FUNCTION_BLOCK CM_MOVITRAC_B EXTENDS CM_Base //IMPLEMENTS I_Motor_base
VAR_INPUT
	i_stSettings : ST_SettingsMOVITRAC_B_WithBrake;
	i_bIclkForward : BOOL := TRUE; //TRUE = interlocked
	i_bIclkBackward : BOOL := TRUE; //TRUE = interlocked
	
	i_ref_eCtrlState : REFERENCE TO E_CtrlState;
END_VAR
VAR
	// Inputs
	I_bStaReadyForOperation AT %I* : BOOL; // Drive is ready operation (no error)
	I_bStaMotorIsRunning AT %I* : BOOL; // Drive/motor is running
	
	// Outputs
	Q_bCmdReset AT %Q* : BOOL; // Command to reset drive.
	Q_bCmdEnable AT %Q* : BOOL; // Command to enable drive.
	Q_bCmdStartCW AT %Q* : BOOL; // Command start in clock-wise direction.
	Q_bCmdStartCCW AT %Q* : BOOL; // Command start in counter-clock-wise direction.
	
	Q_bCmdReleaseBrake AT %Q* : BOOL; // Command to release brake
	Q_nSetTargetSpeed AT %Q* : INT; // Target speed
	
	// Force outputs (IO-test functions)
	s_fbForceCmdReset : FB_ForceOutput;
	s_fbForceCmdEnable : FB_ForceOutput;
	s_fbForceCmdStartCW : FB_ForceOutput;
	s_fbForceCmdStartCCW : FB_ForceOutput;
	s_fbForceCmdReleaseBrake : FB_ForceOutput;
	s_fForceValueTargetSpeed : LREAL; //[0..100%]
	
	//Interlocks
	s_bIclkForward : BOOL;
	s_bIclkBackward : BOOL;
	
	// Requests
	s_bReqStop : BOOL;
	s_bReqStartForward : BOOL;
	s_bReqStartBackward : BOOL;
	s_bReqReleaseBrake : BOOL;
	s_bReqApplyBrake : BOOL;
	s_bReqReset : BOOL;
	
	// Commands
	s_bCmdEnable : BOOL;
	s_bCmdReset : BOOL;
	s_bCmdForward : BOOL;
	s_bCmdBackward : BOOL;
	s_bCmdReleaseBrake : BOOL;
		
	// States
	s_bStaReadyForOperation: BOOL;
	s_bStaDriveError: BOOL;
	s_bStaBrakeReleased : BOOL;
	s_bStaMotorStopped : BOOL;
	s_bStaWarning : BOOL;
	
	s_sInterlockedReasonForward : STRING; //External interlocked reason for clarifying reason
	s_sInterlockedReasonBackward : STRING; //External interlocked reason for clarifying reason
	
	// Setpoints
	s_fTargetSpeed : LREAL; // Target speed [mm/s]
	
	// Timers
	s_tofResetPulse : TOF;
	s_tonMotorStoppedDelay : TON;
	s_tonBrakeReleasedDelay : TON;
	
	// Alarms
	s_fbAlarmHandlerDriveError : FB_AlarmHandler;
	s_fbAlarmHandlerApplyingBrakeNotAllowed : FB_AlarmHandler;
	s_fbAlarmHandlerStartMotorNotAllowed : FB_AlarmHandler;
	s_fbAlarmHandlerMotorForwardInterlocked : FB_AlarmHandler;
	s_fbAlarmHandlerMotorBackwardInterlocked : FB_AlarmHandler;
	
	s_errDriveError : BOOL;
	s_wrnApplyingBrakeNotAllowed : BOOL;
	s_wrnStartMotorNotAllowed : BOOL;
	s_wrnMotorForwardInterlocked : BOOL;
	s_wrnMotorBackwardInterlocked : BOOL;
	
	//Hmi
	s_fbHmiBtnManualReleaseBrake: FB_HmiBtn;
	s_fbHmiBtnManualApplyBrake	: FB_HmiBtn;
	s_fbHmiBtnManualForward		: FB_HmiBtn;
	s_fbHmiBtnManualBackward	: FB_HmiBtn;
	s_fbHmiBtnManualStop		: FB_HmiBtn;
	s_fbHmiBtnManualReset		: FB_HmiBtn;
	
	s_fbHmiLedBrakeReleased		: FB_HmiLed;
	s_fbHmiLedMotorStopped		: FB_HmiLed;
	s_fbHmiLedDriveError		: FB_HmiLed;
	
	//Sequence
	eSeqMOVITRAC_B_WithBrake : E_SeqMOVITRAC_B_WithBrake;
	seqTimer : TON;
	seqPreStep : E_SeqMOVITRAC_B_WithBrake;
	s_sActStep : STRING;
	
END_VAR

VAR CONSTANT
	cMAX_INT_VALUE : INT := 32767;
END_VAR


SUPER^();

METHOD PROTECTED _m_Alarms : BOOL

IF NOT SUPER^._m_Alarms() THEN
	RETURN;
END_IF

// Set error bits
s_errDriveError := i_bReqEnable AND s_bStaDriveError;// AND NOT(i_bCmdReset);

// Interlock warnings
IF s_bIclkForward AND NOT(s_bStaMotorStopped) THEN	
	s_wrnMotorForwardInterlocked := TRUE;
	m_Stop();
ELSIF NOT(s_bIclkForward) OR i_bCmdReset THEN
	s_wrnMotorForwardInterlocked := FALSE;
END_IF

IF s_bIclkBackward AND NOT(s_bStaMotorStopped) THEN
	s_wrnMotorBackwardInterlocked := TRUE;
	m_Stop();
ELSIF NOT(s_bIclkBackward) OR i_bCmdReset THEN
	s_wrnMotorBackwardInterlocked := FALSE;
END_IF

// Alarm Handlers
s_fbAlarmHandlerDriveError(
	i_bStaActive := s_errDriveError,
	i_eAlarmLevel := E_AlarmLevel.Alarm,
	i_sAlarmText := CONCAT(i_sCmName, ': Drive - has error (check drive).'));
	
s_fbAlarmHandlerApplyingBrakeNotAllowed(
	i_bStaActive := s_wrnApplyingBrakeNotAllowed,
	i_eAlarmLevel := E_AlarmLevel.Warning,
	i_sAlarmText := CONCAT(i_sCmName, ': Brake - not allowed to be applied (motor not stopped).'));
	
s_wrnApplyingBrakeNotAllowed R= s_bStaMotorStopped;
	
s_fbAlarmHandlerStartMotorNotAllowed(
	i_bStaActive := s_wrnStartMotorNotAllowed,
	i_eAlarmLevel := E_AlarmLevel.Warning,
	i_sAlarmText := CONCAT(i_sCmName, ': Motor - not allowed to start (brake not released).'));
	
s_wrnStartMotorNotAllowed R= s_bStaBrakeReleased;
	
s_fbAlarmHandlerMotorForwardInterlocked(
	i_bStaActive := s_wrnMotorForwardInterlocked,
	i_eAlarmLevel := E_AlarmLevel.Warning,
	i_sAlarmText := CONCAT(i_sCmName, CONCAT(': Motor - interlocked to move forward, Reason: ',CONCAT(s_sInterlockedReasonForward, '.'))));
	//--i_sAlarmText := CONCAT(i_sCmName, CONCAT(': Motor - interlocked to move forward, Reason: ',CONCAT(i_fbInterlockConvFwd.p_sReason, '.'))));
	
s_fbAlarmHandlerMotorBackwardInterlocked(
	i_bStaActive := s_wrnMotorBackwardInterlocked,
	i_eAlarmLevel := E_AlarmLevel.Warning,
	i_sAlarmText := CONCAT(i_sCmName, CONCAT(': Motor - interlocked to move backward, Reason: ',CONCAT(s_sInterlockedReasonBackward, '.'))));
	//--i_sAlarmText := CONCAT(i_sCmName, CONCAT(': Motor - interlocked to move backward, Reason: ',CONCAT(i_fbInterlockConvBwd.p_sReason, '.'))));
	
// Alarm collector	
s_bStaError := 
	s_fbAlarmHandlerDriveError.q_bStaActive;

// Warning collector
s_bStaWarning := 
	s_fbAlarmHandlerApplyingBrakeNotAllowed.q_bStaActive
	OR s_fbAlarmHandlerStartMotorNotAllowed.q_bStaActive
	OR s_fbAlarmHandlerMotorForwardInterlocked.q_bStaActive
	OR s_fbAlarmHandlerMotorBackwardInterlocked.q_bStaActive;	
	
_m_Alarms := TRUE;
END_METHOD

METHOD PROTECTED _m_Devices : BOOL

IF NOT SUPER^._m_Devices() THEN
	RETURN;
END_IF

//Exception error
IF (s_bStaError OR NOT(i_bReqEnable))
	AND (eSeqMOVITRAC_B_WithBrake < E_SeqMOVITRAC_B_WithBrake.STOPPING) THEN
		eSeqMOVITRAC_B_WithBrake := E_SeqMOVITRAC_B_WithBrake.STOPPING;
END_IF 

seqTimer(
	IN := (eSeqMOVITRAC_B_WithBrake = seqPreStep),
	PT := T#3600S);
	
seqPreStep := eSeqMOVITRAC_B_WithBrake;

s_sActStep := TO_STRING(eSeqMOVITRAC_B_WithBrake);
	
CASE eSeqMOVITRAC_B_WithBrake OF
	
	E_SeqMOVITRAC_B_WithBrake.INIT:
		_m_ResetAllRequests();
	
		//Reset commands
		s_bCmdForward := FALSE;
		s_bCmdBackward := FALSE;	
		s_bCmdReleaseBrake := FALSE;
		s_bCmdReset := FALSE;
		s_bCmdEnable := FALSE;
		s_fTargetSpeed := 0;
		
		//Reset states
		s_bStaBrakeReleased := FALSE;
		s_bStaDriveError := FALSE;
		//s_bStaMotorStopped := FALSE;			written by inputs()
		//s_bStaReadyForOperation := FALSE;		written by inputs()
	
		eSeqMOVITRAC_B_WithBrake := E_SeqMOVITRAC_B_WithBrake.STOPPED; 
		
	E_SeqMOVITRAC_B_WithBrake.STOPPED:
		s_bStaBrakeReleased := FALSE;
		//--s_bStaMotorStopped := TRUE;			written by inputs()
		s_bReqStop := FALSE;
		s_bStaReadyForOperation := TRUE;
		
		IF (s_bReqReleaseBrake OR s_bReqStartForward OR s_bReqStartBackward) THEN
			eSeqMOVITRAC_B_WithBrake := E_SeqMOVITRAC_B_WithBrake.RELEASE_BRAKE;
		END_IF

		IF s_bReqApplyBrake THEN
			eSeqMOVITRAC_B_WithBrake := E_SeqMOVITRAC_B_WithBrake.APPLY_BRAKE;
		END_IF
		
		IF seqTimer.PT >= T#10S THEN
			s_bCmdEnable := FALSE;
		END_IF
			
	E_SeqMOVITRAC_B_WithBrake.RELEASE_BRAKE:
		s_bCmdReleaseBrake := TRUE;
		s_bReqReleaseBrake := FALSE;
		
		IF seqTimer.ET > i_stSettings.tBrakeReleasedDelay THEN
			s_bStaBrakeReleased := TRUE;
		END_IF
		
		IF s_bReqStop THEN
			eSeqMOVITRAC_B_WithBrake := E_SeqMOVITRAC_B_WithBrake.STOPPING;
		ELSIF s_bStaBrakeReleased AND s_bReqStartForward THEN
			s_bCmdEnable := TRUE;
			eSeqMOVITRAC_B_WithBrake := E_SeqMOVITRAC_B_WithBrake.MOVING_FORWARD;
		ELSIF s_bStaBrakeReleased AND s_bReqStartBackward THEN
			s_bCmdEnable := TRUE;
			eSeqMOVITRAC_B_WithBrake := E_SeqMOVITRAC_B_WithBrake.MOVING_BACKWARD;
		ELSIF s_bReqApplyBrake THEN
			eSeqMOVITRAC_B_WithBrake := E_SeqMOVITRAC_B_WithBrake.APPLY_BRAKE;
		END_IF
	
	E_SeqMOVITRAC_B_WithBrake.MOVING_FORWARD:
		s_bCmdForward := TRUE;
		s_bReqStartForward := FALSE;
		
		//--s_bStaMotorStopped := FALSE;		written by inputs()
		//s_fTargetSpeed is written by method 
	
		IF s_bReqStop THEN
			eSeqMOVITRAC_B_WithBrake := E_SeqMOVITRAC_B_WithBrake.STOPPING;
		END_IF
		
	E_SeqMOVITRAC_B_WithBrake.MOVING_BACKWARD:
		s_bCmdBackward := TRUE;
		s_bReqStartBackward := FALSE;
		
		//--s_bStaMotorStopped := FALSE;		//written by inputs()
		//s_fTargetSpeed is written by method 
	
		IF s_bReqStop THEN
			eSeqMOVITRAC_B_WithBrake := E_SeqMOVITRAC_B_WithBrake.STOPPING;
		END_IF
	
	E_SeqMOVITRAC_B_WithBrake.STOPPING:
		s_bCmdForward := FALSE;
		s_bCmdBackward := FALSE;
		s_bReqStop := FALSE;
		
		IF s_bStaMotorStopped THEN
			eSeqMOVITRAC_B_WithBrake := E_SeqMOVITRAC_B_WithBrake.APPLY_BRAKE;
		END_IF
		
		//--IF seqTimer.ET > i_stSettings.tMotorStoppedDelay THEN
			//--s_bStaMotorStopped := TRUE;		//Written by inputs()
			//--eSeqMOVITRAC_B_WithBrake := E_SeqMOVITRAC_B_WithBrake.APPLY_BRAKE;
		//--END_IF	
	
	E_SeqMOVITRAC_B_WithBrake.APPLY_BRAKE:
		s_bCmdReleaseBrake := FALSE;
		s_bReqApplyBrake := FALSE;
		
		IF seqTimer.ET > i_stSettings.tBrakeReleasedDelay THEN
			s_bStaBrakeReleased := FALSE;
			
			IF (s_bStaError OR NOT(i_bReqEnable)) THEN
				eSeqMOVITRAC_B_WithBrake := E_SeqMOVITRAC_B_WithBrake.ERROR;
			ELSE
				_m_ResetAllRequests();
				eSeqMOVITRAC_B_WithBrake := E_SeqMOVITRAC_B_WithBrake.STOPPED;
			END_IF	
		END_IF
		
	E_SeqMOVITRAC_B_WithBrake.ERROR:
		s_bCmdReset := i_bCmdReset OR s_bReqReset;
		s_bReqReset := FALSE;
		
		IF (NOT(s_bStaError) AND i_bReqEnable) THEN
			eSeqMOVITRAC_B_WithBrake := E_SeqMOVITRAC_B_WithBrake.INIT;
		END_IF
		
END_CASE

_m_Devices := TRUE;
END_METHOD

METHOD PROTECTED _m_Hmi : BOOL

IF NOT SUPER^._m_Hmi() THEN
	RETURN;
END_IF

//Buttons
s_fbHmiBtnManualReleaseBrake();
s_fbHmiBtnManualApplyBrake();
s_fbHmiBtnManualForward();
s_fbHmiBtnManualBackward();
s_fbHmiBtnManualStop();
s_fbHmiBtnManualReset();

//Led
s_fbHmiLedBrakeReleased(i_bStaLed := s_bStaBrakeReleased);
s_fbHmiLedMotorStopped(i_bStaLed := s_bStaMotorStopped);
s_fbHmiLedDriveError(i_bStaLed := s_bStaDriveError);
(*
{warning '#TODO: Add manual control from hmi'}
CASE i_eCtrlMode OF

	E_CtrlMode.IDLE..
	E_CtrlMode.AUTOMATIC:
		s_fbHmiBtnManualReleaseBrake.p_bStaVisible := FALSE;
		s_fbHmiBtnManualReleaseBrake.p_bStaEnabled := FALSE;
		
		s_fbHmiBtnManualApplyBrake.p_bStaVisible := FALSE;
		s_fbHmiBtnManualApplyBrake.p_bStaEnabled := FALSE;
		
		s_fbHmiBtnManualForward.p_bStaVisible := FALSE;
		s_fbHmiBtnManualForward.p_bStaEnabled := FALSE;
		
		s_fbHmiBtnManualBackward.p_bStaVisible := FALSE;
		s_fbHmiBtnManualBackward.p_bStaEnabled := FALSE;
		
		s_fbHmiBtnManualStop.p_bStaVisible := FALSE;
		s_fbHmiBtnManualStop.p_bStaEnabled := FALSE;
		
		s_fbHmiBtnManualReset.p_bStaVisible := FALSE;
		s_fbHmiBtnManualReset.p_bStaEnabled := FALSE;
	
	E_CtrlMode.MANUAL:
		//Is het de bedoeling om op deze plekken de hmi knoppen aan te sturen, OF moet dat gedaan worden in METHOD hmi?
		s_fbHmiBtnManualReleaseBrake.p_bStaVisible := TRUE;
		s_fbHmiBtnManualReleaseBrake.p_bStaEnabled := i_bReqEnable;
		
		s_fbHmiBtnManualApplyBrake.p_bStaVisible := TRUE;
		s_fbHmiBtnManualApplyBrake.p_bStaEnabled := i_bReqEnable AND s_bStaMotorStopped;
		
		s_fbHmiBtnManualForward.p_bStaVisible := TRUE;
		s_fbHmiBtnManualForward.p_bStaEnabled := i_bReqEnable AND s_bStaMotorStopped (*AND s_bStaBrakeReleased*) AND NOT(i_bIclkForward);
		
		s_fbHmiBtnManualBackward.p_bStaVisible := TRUE;
		s_fbHmiBtnManualBackward.p_bStaEnabled := i_bReqEnable AND s_bStaMotorStopped (*AND s_bStaBrakeReleased*) AND NOT(i_bIclkBackward);
		
		s_fbHmiBtnManualStop.p_bStaVisible := TRUE;
		s_fbHmiBtnManualStop.p_bStaEnabled := TRUE;
		
		s_fbHmiBtnManualReset.p_bStaVisible := TRUE;
		s_fbHmiBtnManualReset.p_bStaEnabled := TRUE;
		
		IF s_fbHmiBtnManualReleaseBrake.p_osrBtnPress THEN
			m_ReleaseBrake();
		END_IF
	
		IF s_fbHmiBtnManualApplyBrake.p_osrBtnPress THEN
			m_ApplyBrake();
		END_IF
			
		IF s_fbHmiBtnManualStop.p_osrBtnPress THEN
			m_Stop();	
		ELSIF s_fbHmiBtnManualForward.p_osrBtnPress THEN
			m_StartForward(i_rTargetSpeed := s_fTargetSpeed);
		ELSIF s_fbHmiBtnManualBackward.p_osrBtnPress THEN
			m_StartBackward(i_rTargetSpeed := s_fTargetSpeed);
		END_IF

		IF s_fbHmiBtnManualReset.p_osrBtnPress THEN
			m_Reset();
		END_IF	
	
END_CASE
*)
IF __ISVALIDREF(i_ref_eCtrlState) THEN
	//MAINTENANCE-mode is running
	IF (i_eCtrlMode = E_CtrlMode.MAINTENANCE) AND (i_ref_eCtrlState = E_CtrlState.RUNNING) THEN
		s_fbHmiBtnManualReleaseBrake.p_bStaVisible := TRUE;
		s_fbHmiBtnManualReleaseBrake.p_bStaEnabled := i_bReqEnable;
		
		s_fbHmiBtnManualApplyBrake.p_bStaVisible := TRUE;
		s_fbHmiBtnManualApplyBrake.p_bStaEnabled := i_bReqEnable AND s_bStaMotorStopped;
		
		s_fbHmiBtnManualForward.p_bStaVisible := TRUE;
		s_fbHmiBtnManualForward.p_bStaEnabled := i_bReqEnable AND s_bStaMotorStopped (*AND s_bStaBrakeReleased*) AND NOT(i_bIclkForward);
		
		s_fbHmiBtnManualBackward.p_bStaVisible := TRUE;
		s_fbHmiBtnManualBackward.p_bStaEnabled := i_bReqEnable AND s_bStaMotorStopped (*AND s_bStaBrakeReleased*) AND NOT(i_bIclkBackward);
		
		s_fbHmiBtnManualStop.p_bStaVisible := TRUE;
		s_fbHmiBtnManualStop.p_bStaEnabled := TRUE;
		
		s_fbHmiBtnManualReset.p_bStaVisible := TRUE;
		s_fbHmiBtnManualReset.p_bStaEnabled := TRUE;
		
		IF s_fbHmiBtnManualReleaseBrake.p_osrBtnPress THEN
			m_ReleaseBrake();
		END_IF
	
		IF s_fbHmiBtnManualApplyBrake.p_osrBtnPress THEN
			m_ApplyBrake();
		END_IF
			
		IF s_fbHmiBtnManualStop.p_osrBtnPress THEN
			m_Stop();	
		ELSIF s_fbHmiBtnManualForward.p_osrBtnPress THEN
			m_StartForward(i_rTargetSpeed := s_fTargetSpeed);
		ELSIF s_fbHmiBtnManualBackward.p_osrBtnPress THEN
			m_StartBackward(i_rTargetSpeed := s_fTargetSpeed);
		END_IF

		IF s_fbHmiBtnManualReset.p_osrBtnPress THEN
			m_Reset();
		END_IF
		
	//other-mode	
	ELSE
		s_fbHmiBtnManualReleaseBrake.p_bStaVisible := FALSE;
		s_fbHmiBtnManualReleaseBrake.p_bStaEnabled := FALSE;
		
		s_fbHmiBtnManualApplyBrake.p_bStaVisible := FALSE;
		s_fbHmiBtnManualApplyBrake.p_bStaEnabled := FALSE;
		
		s_fbHmiBtnManualForward.p_bStaVisible := FALSE;
		s_fbHmiBtnManualForward.p_bStaEnabled := FALSE;
		
		s_fbHmiBtnManualBackward.p_bStaVisible := FALSE;
		s_fbHmiBtnManualBackward.p_bStaEnabled := FALSE;
		
		s_fbHmiBtnManualStop.p_bStaVisible := FALSE;
		s_fbHmiBtnManualStop.p_bStaEnabled := FALSE;
		
		s_fbHmiBtnManualReset.p_bStaVisible := FALSE;
		s_fbHmiBtnManualReset.p_bStaEnabled := FALSE;
	END_IF
END_IF
	
_m_Hmi := TRUE;
END_METHOD

METHOD PROTECTED _m_Init : BOOL

IF NOT SUPER^._m_Init() THEN
	RETURN;
END_IF

{warning '#TODO: Not sure if this control module needs initialzation'}
//--s_DOValve.i_stSettings.bCfgDelay 		:= FALSE;
//--s_DOValve.i_stSettings.tmOutputDelay 	:= T#0S;

//Hmi 
	s_fbHmiBtnManualReleaseBrake.p_eButtontype := E_HmiButtonType.PUSHBUTTON;
	s_fbHmiBtnManualReleaseBrake.p_bStaVisible := FALSE;
	s_fbHmiBtnManualReleaseBrake.p_bStaEnabled := FALSE;		
	s_fbHmiBtnManualReleaseBrake.p_sBtnText := 'Release Brake';
	
	s_fbHmiBtnManualApplyBrake.p_eButtontype := E_HmiButtonType.PUSHBUTTON;
	s_fbHmiBtnManualApplyBrake.p_bStaVisible := FALSE;
	s_fbHmiBtnManualApplyBrake.p_bStaEnabled := FALSE;		
	s_fbHmiBtnManualApplyBrake.p_sBtnText := 'Apply Brake';
	
	s_fbHmiBtnManualForward.p_eButtontype := E_HmiButtonType.PUSHBUTTON;
	s_fbHmiBtnManualForward.p_bStaVisible := FALSE;
	s_fbHmiBtnManualForward.p_bStaEnabled := FALSE;		
	s_fbHmiBtnManualForward.p_sBtnText := 'Move Forward';
	
	s_fbHmiBtnManualBackward.p_eButtontype := E_HmiButtonType.PUSHBUTTON;
	s_fbHmiBtnManualBackward.p_bStaVisible := FALSE;
	s_fbHmiBtnManualBackward.p_bStaEnabled := FALSE;		
	s_fbHmiBtnManualBackward.p_sBtnText := 'Move Backward';
	
	s_fbHmiBtnManualStop.p_eButtontype := E_HmiButtonType.PUSHBUTTON;
	s_fbHmiBtnManualStop.p_bStaVisible := FALSE;
	s_fbHmiBtnManualStop.p_bStaEnabled := FALSE;		
	s_fbHmiBtnManualStop.p_sBtnText := 'Stop';

	s_fbHmiBtnManualReset.p_eButtontype := E_HmiButtonType.PUSHBUTTON;
	s_fbHmiBtnManualReset.p_bStaVisible := FALSE;
	s_fbHmiBtnManualReset.p_bStaEnabled := FALSE;		
	s_fbHmiBtnManualReset.p_sBtnText := 'Reset';
	
	s_fbHmiLedBrakeReleased.p_bStaVisible := FALSE;
	s_fbHmiLedBrakeReleased.p_sToHmiDescriptionLed := 'Brake Released';
	
	s_fbHmiLedMotorStopped.p_bStaVisible := FALSE;
	s_fbHmiLedMotorStopped.p_sToHmiDescriptionLed := 'Motor Stopped';
	
	s_fbHmiLedDriveError.p_bStaVisible := FALSE;
	s_fbHmiLedDriveError.p_sToHmiDescriptionLed := 'Drive Error';
	
_m_Init := TRUE;
END_METHOD

METHOD PROTECTED _m_Inputs : BOOL

IF NOT SUPER^._m_Inputs() THEN
	RETURN;
END_IF

s_bStaReadyForOperation := I_bStaReadyForOperation;
s_bStaDriveError := NOT(I_bStaReadyForOperation);
s_bStaMotorStopped := NOT(I_bStaMotorIsRunning);

s_bIclkForward := i_bIclkForward;
s_bIclkBackward := i_bIclkBackward;

//--s_bIclkForward := i_fbInterlockConvFwd.p_bInterlocked;
//--s_bIclkBackward := i_fbInterlockConvBwd.p_bInterlocked;

_m_Inputs := TRUE;
END_METHOD

METHOD PROTECTED _m_Outputs : BOOL

IF NOT SUPER^._m_Outputs() THEN
	RETURN;
END_IF

{warning #TODO: Nog bepalen OF het beter is om onderstaande code te verwerken in FB_Force output}
IF __ISVALIDREF(i_ref_eCtrlState) THEN
	IF (i_eCtrlMode <> E_CtrlMode.IO) OR (i_ref_eCtrlState <> E_CtrlState.RUNNING) THEN
		s_fbForceCmdEnable.i_eForceValue := E_ForceValue.RELEASED;
		s_fbForceCmdReset.i_eForceValue := E_ForceValue.RELEASED;
		s_fbForceCmdStartCW.i_eForceValue := E_ForceValue.RELEASED;
		s_fbForceCmdStartCCW.i_eForceValue := E_ForceValue.RELEASED;
		s_fbForceCmdReleaseBrake.i_eForceValue := E_ForceValue.RELEASED;
		s_fForceValueTargetSpeed := 0.0;
	END_IF
END_IF 

s_fbForceCmdEnable(
	i_ref_bCmdInput := s_bCmdEnable,
	i_ref_bCmdOutput := Q_bCmdEnable);
	
s_fbForceCmdReset(
	i_ref_bCmdInput := s_bCmdReset,
	i_ref_bCmdOutput := Q_bCmdReset);
	
s_fbForceCmdStartCW(
	i_ref_bCmdInput := s_bCmdForward,
	i_ref_bCmdOutput := Q_bCmdStartCW);
	
s_fbForceCmdStartCCW(
	i_ref_bCmdInput := s_bCmdBackward,
	i_ref_bCmdOutput := Q_bCmdStartCCW);
	
s_fbForceCmdReleaseBrake(
	i_ref_bCmdInput := s_bCmdReleaseBrake,
	i_ref_bCmdOutput := Q_bCmdReleaseBrake);

IF s_fForceValueTargetSpeed = 0.0 THEN
	Q_nSetTargetSpeed := LREAL_TO_INT(s_fTargetSpeed / i_stSettings.rMaxTargetSpeed * cMAX_INT_VALUE); // [mm/s]
ELSE	
	Q_nSetTargetSpeed := LREAL_TO_INT(s_fForceValueTargetSpeed / 100.0  * cMAX_INT_VALUE); // [%]
END_IF 
	
_m_Outputs := TRUE;
END_METHOD

METHOD PRIVATE _m_ResetAllRequests

s_bReqStop :=
s_bReqStartForward :=
s_bReqStartBackward :=
s_bReqReleaseBrake :=
s_bReqApplyBrake :=
s_bReqReset := FALSE;
END_METHOD

METHOD PUBLIC m_ApplyBrake : BOOL

IF NOT i_bReqEnable THEN 
	RETURN;
END_IF

s_bReqApplyBrake := TRUE;

m_ApplyBrake := NOT(s_bStaBrakeReleased);
END_METHOD

/// Release brake
METHOD PUBLIC m_ReleaseBrake : BOOL

IF NOT i_bReqEnable THEN 
	RETURN;
END_IF

s_bReqReleaseBrake := TRUE;

m_ReleaseBrake := s_bStaBrakeReleased;
END_METHOD

METHOD PUBLIC m_Reset : BOOL

IF NOT i_bReqEnable THEN 
	RETURN;
END_IF

s_bReqReset := TRUE;

m_Reset := s_bCmdReset;
END_METHOD

METHOD PUBLIC m_StartBackward : BOOL
VAR_INPUT
	i_rTargetSpeed : LREAL; // Target speed [mm/s]
END_VAR

IF NOT i_bReqEnable THEN 
	RETURN;
END_IF

//--IF NOT(i_bIclkBackward) THEN
//--IF NOT(i_fbInterlockConvBwd.p_bInterlocked) THEN
IF NOT(s_bIclkBackward) THEN
	s_bReqStartBackward := TRUE;
	
	IF i_rTargetSpeed < 0 THEN
		s_fTargetSpeed := 0;
	ELSIF i_rTargetSpeed > cMAX_INT_VALUE THEN	
		i_rTargetSpeed := cMAX_INT_VALUE;
	ELSE 
		s_fTargetSpeed := i_rTargetSpeed;
	END_IF
	
ELSE
	s_wrnMotorBackwardInterlocked := TRUE;
END_IF

m_StartBackward := s_bCmdBackward;
END_METHOD

METHOD PUBLIC m_StartForward : BOOL
VAR_INPUT
	i_rTargetSpeed : LREAL; // Target speed [mm/s]
END_VAR

IF NOT i_bReqEnable THEN 
	RETURN;
END_IF

IF NOT(s_bIclkForward) THEN
	s_bReqStartForward := TRUE;
	
	IF i_rTargetSpeed < 0 THEN
		s_fTargetSpeed := 0;
	ELSIF i_rTargetSpeed > cMAX_INT_VALUE THEN	
		i_rTargetSpeed := cMAX_INT_VALUE;
	ELSE 
		s_fTargetSpeed := i_rTargetSpeed;
	END_IF
	
ELSE	
	s_wrnMotorForwardInterlocked := TRUE;
END_IF

m_StartForward := s_bCmdForward;
END_METHOD

METHOD PUBLIC m_Stop : BOOL

IF NOT i_bReqEnable THEN 
	RETURN;
END_IF

s_bReqStop := TRUE;

m_Stop := s_bStaMotorStopped;
END_METHOD

{attribute 'monitoring':='call'}
PROPERTY PUBLIC p_bStaBrakeReleased : BOOL
GET

p_bStaBrakeReleased := s_bStaBrakeReleased;
END_GET
END_PROPERTY

{attribute 'monitoring':='call'}
PROPERTY PUBLIC p_bStaMotorRunning : BOOL
GET

p_bStaMotorRunning := s_bStaReadyForOperation AND NOT(s_bStaMotorStopped);
END_GET
END_PROPERTY

{attribute 'monitoring':='call'}
PROPERTY PUBLIC p_bStaMotorStopped : BOOL
GET

p_bStaMotorStopped := s_bStaMotorStopped;
END_GET
END_PROPERTY

{attribute 'monitoring':='call'}
PROPERTY PUBLIC p_bStaWarning : BOOL
GET

p_bStaWarning := s_bStaWarning;
END_GET
END_PROPERTY

{attribute 'monitoring':='call'}
PROPERTY PUBLIC p_sInterlockedReasonBackward : STRING(GVL.g_MAX_LEN_INTERLOCK_REASON)
GET

p_sInterlockedReasonBackward := s_sInterlockedReasonBackward;
END_GET
SET

s_sInterlockedReasonBackward := p_sInterlockedReasonBackward;
END_SET
END_PROPERTY

{attribute 'monitoring':='call'}
PROPERTY PUBLIC p_sInterlockedReasonForward : STRING(GVL.g_MAX_LEN_INTERLOCK_REASON)
GET

p_sInterlockedReasonForward := s_sInterlockedReasonForward;
END_GET
SET

s_sInterlockedReasonForward := p_sInterlockedReasonForward;
END_SET
END_PROPERTY

END_FUNCTION_BLOCK

(* stored: Version 1.1.0.1, ProductVersion 3.1.4024.12
   POU CM_MOVITRAC_B: Id {fa9a3c02-fb9e-4f0d-9f6f-ce091f3d4d49}, SpecialFunc None
   Folder Methods: Id {11b83f51-5f87-456d-a35a-77d461c1ecc9}
   Folder Properties: Id {da903959-0eba-44a7-a4b8-91c25055de14}
   Method _m_Alarms: Id {7df04d62-5845-4a1e-8448-72d9b9d8341e}
   Method _m_Devices: Id {5370e1e6-83cf-430a-947c-f21bd2f1ec4b}
   Method _m_Hmi: Id {8b0bfc2b-cd59-45fd-861e-58a9388af400}
   Method _m_Init: Id {10fb3c9f-1aaa-45dc-b899-79bd4e709ce6}
   Method _m_Inputs: Id {e38cdb59-a84f-476e-9954-e5b28d6d08e3}
   Method _m_Outputs: Id {ba15960a-e792-4086-9871-b1105c2a6ed2}
   Method _m_ResetAllRequests: Id {a63c1714-18c0-4e0c-82e9-37ffe0e0464a}
   Method m_ApplyBrake: Id {da833913-48c7-4bfc-979e-1bb75e0dd689}
   Method m_ReleaseBrake: Id {e96b1d6a-c145-4ed0-b15b-db24c9d0f5cd}
   Method m_Reset: Id {c3f29afd-c735-464b-b9f7-dd53b191eb73}
   Method m_StartBackward: Id {3070eb62-39b9-41c5-ab6f-4f29bd1c0220}
   Method m_StartForward: Id {39ee694a-3d82-40c1-89dd-29f4a0ed3ffe}
   Method m_Stop: Id {9f4f7520-546f-4d70-8901-b1fe2259dd85}
   Property p_bStaBrakeReleased: Id {a5ae057d-10d6-4733-b5dd-5152d1849281}
   Get Get: Id {807fee9a-9ade-4c40-8d61-217989029805}
   Property p_bStaMotorRunning: Id {63a7d5b0-0187-4f50-88ae-20969844be04}
   Get Get: Id {3540dc03-69f4-489e-a43f-e10f4335894d}
   Property p_bStaMotorStopped: Id {b36f4974-cbc4-4429-a6eb-dc28eb73aab3}
   Get Get: Id {f5cfef73-d561-4b91-80a5-530b320cf15c}
   Property p_bStaWarning: Id {5b5f03fd-2411-44c8-aae7-3196706a8139}
   Get Get: Id {cd7f0767-6cc8-4566-ac13-1325d1723ac3}
   Property p_sInterlockedReasonBackward: Id {0c7533b0-6229-4bd7-a6ac-beef68a0441b}
   Get Get: Id {89d301ab-99e1-407a-8ad8-3decf2378b91}
   Set Set: Id {f1403b8e-daa5-4ba7-a249-a1171f717224}
   Property p_sInterlockedReasonForward: Id {ee05b23b-0c2f-4ed6-802a-db01c009192a}
   Get Get: Id {d1567d66-dae7-4c45-a522-cf9b9ae0c9db}
   Set Set: Id {232bb7c9-7ead-42b4-a88b-2101a33b73a3} *)
